{region '#Template'}
	{attribute 'Category' := 'Universal'}
	{attribute 'Version' := '0.0.1.0'}
	{attribute 'Tags' := 'Universal, Control, Timer switch-on delayed'}
	{attribute 'Description' := 'Zeitglied Einschaltverzögert	// Timer switch-on delayed'}
{endregion}
FUNCTION_BLOCK FB_BA_DlyOn EXTENDS FB_BA_View
VAR_INPUT
	bVal					: BOOL;	
END_VAR
VAR_OUTPUT
	bQ						: BOOL;	
END_VAR
VAR_INPUT CONSTANT
	TiDly					: FB_BA_AV_Op;		
END_VAR	
VAR	
	tofDlyOn				: TON;
END_VAR
VAR // added by the converter: edge detectors and wires of the graphical bodies
    _w1 : ANY;
END_VAR

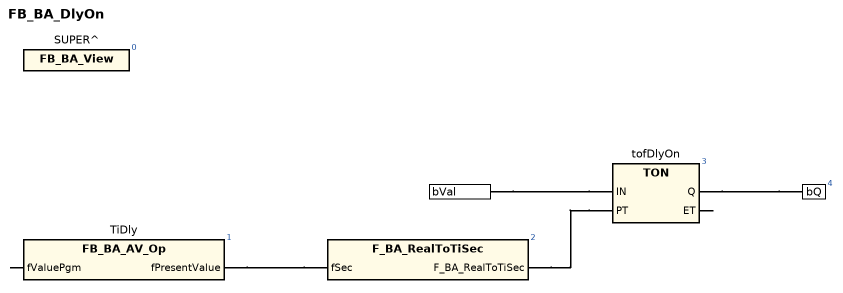
SUPER^(); // FB_BA_View
TiDly(); // FB_BA_AV_Op
_w1 := F_BA_RealToTiSec(fSec := TiDly.fPresentValue);
tofDlyOn(IN := bVal, PT := _w1); // TON
bQ := tofDlyOn.Q;

METHOD FB_init : BOOL
VAR_INPUT
	bInitRetains : BOOL; // if TRUE, the retain variables are initialized (warm start / cold start)
	bInCopyCode : BOOL;  // if TRUE, the instance afterwards gets moved into the copy code (online change)
END_VAR
TiDly.iParent			:= THIS^;
TiDly.iLabel			:= LblUniControl.DelayOn_TiDly;		 
TiDly.sObjectName		:= '{Idx=01}';								 	 
TiDly.eUnit 			:= E_BA_Unit.eTime_Seconds;								 
TiDly.fValueRm			:= 0;		
TiDly.fCOVIncrement		:= BA2_Param.fDefCOVIncrement;
END_METHOD

END_FUNCTION_BLOCK

(* stored: Version 1.1.0.1, ProductVersion 3.1.4024.6
   POU FB_BA_DlyOn: Id {bf448dfa-89af-4802-95ed-458d49c7ae8b}, SpecialFunc None
   Method FB_init: Id {00cc2adc-40dd-4c51-9fd1-7e8123212515} *)
